        $ 1403 "Direction: Base Z+"
        global move_thread_flag_1403=0
        thread move_thread_1403():
          enter_critical
          move_thread_flag_1403 = 1
          local towardsPos=calculate_point_to_move_towards(p[0.0,0.0,0.0,0.0,0.0,0.0], [0.0,0.0,1.0], 0.05)
          movel(towardsPos, a=0.04, v=0.03)
          move_thread_flag_1403 = 2
          exit_critical
        end
        move_thread_flag_1403 = 0
        move_thread_han_1403 = run move_thread_1403()
        while (True):
          sleep(1.0E-10)
          if (move_thread_flag_1403 > 1):
            join move_thread_han_1403
            $ 1404 "Until (distance)"
            break
          end
          sync()
        end
        $ 1405 "MoveJ"
        $ 1406 "internos" "breakAfter"
        movej(internos, a=1.3962634015954636, v=1.0471975511965976)
        $ 1407 "Wait: 0.3"
        sleep(0.3)
        $ 1408 "Set CO[1]=Apagar"
        set_configurable_digital_out(1, False)
        $ 1409 "Wait: 0.3"
        sleep(0.3)
        $ 1410 "If barrenoActual≟13"
        if (barrenoActual == 13):
          $ 1411 "Direction: Base Z+"
          global move_thread_flag_1411=0
          thread move_thread_1411():
            enter_critical
            move_thread_flag_1411 = 1
            local towardsPos=calculate_point_to_move_towards(p[0.0,0.0,0.0,0.0,0.0,0.0], [0.0,0.0,1.0], 0.03)
            movel(towardsPos, a=1.2, v=0.25)
            move_thread_flag_1411 = 2
            exit_critical
          end
          move_thread_flag_1411 = 0
          move_thread_han_1411 = run move_thread_1411()
          while (True):
            sleep(1.0E-10)
            if (move_thread_flag_1411 > 1):
              join move_thread_han_1411
              $ 1412 "Until (distance)"
              break
            end
            sync()
          end
          $ 1413 "MoveJ"
          $ 1414 "Zona_izq1" "breakAfter"
          movej(get_inverse_kin(Zona_izq1_p, qnear=Zona_izq1_q), a=1.3962634015954636, v=1.0471975511965976)
          $ 1415 "Posicion_Cero" "breakAfter"
          movej(get_inverse_kin(Posicion_Cero_p, qnear=Posicion_Cero_q), a=1.3962634015954636, v=1.0471975511965976)
          $ 1416 "Call Quitar_Broca_Chida"
          Quitar_Broca_Chida()
          $ 1417 "Call Poner_Broca"
          Poner_Broca()
          $ 1418 "MoveJ"
          $ 1419 "Posicion_Cero" "breakAfter"
          movej(get_inverse_kin(Posicion_Cero_p, qnear=Posicion_Cero_q), a=1.3962634015954636, v=1.0471975511965976)
          $ 1420 "Zona_izq1" "breakAfter"
          movej(get_inverse_kin(Zona_izq1_p, qnear=Zona_izq1_q), a=1.3962634015954636, v=1.0471975511965976)
        else:
          $ 1421 "ElseIf barrenoActual≟27"
          if (barrenoActual == 27):
            $ 1422 "Direction: Base Z+"
            global move_thread_flag_1422=0
            thread move_thread_1422():
              enter_critical
              move_thread_flag_1422 = 1
              local towardsPos=calculate_point_to_move_towards(p[0.0,0.0,0.0,0.0,0.0,0.0], [0.0,0.0,1.0], 0.03)
              movel(towardsPos, a=1.2, v=0.25)
              move_thread_flag_1422 = 2
              exit_critical
            end
            move_thread_flag_1422 = 0
            move_thread_han_1422 = run move_thread_1422()
            while (True):
              sleep(1.0E-10)
              if (move_thread_flag_1422 > 1):
                join move_thread_han_1422
                $ 1423 "Until (distance)"
                break
              end
              sync()
            end
            $ 1424 "MoveJ"
            $ 1425 "Zona_izq1" "breakAfter"
            movej(get_inverse_kin(Zona_izq1_p, qnear=Zona_izq1_q), a=1.3962634015954636, v=1.0471975511965976)
            $ 1426 "Posicion_Cero" "breakAfter"
            movej(get_inverse_kin(Posicion_Cero_p, qnear=Posicion_Cero_q), a=1.3962634015954636, v=1.0471975511965976)
            $ 1427 "Call Quitar_Broca_Chida"
            Quitar_Broca_Chida()
            $ 1428 "Set carrusel_home=Encender"
            modbus_set_output_signal("carrusel_home", True)
            $ 1429 "Wait: 1.0"
            sleep(1.0)
            $ 1430 "Set carrusel_home=Apagar"
            modbus_set_output_signal("carrusel_home", False)
            $ 1431 "Set mensaje_mw10=85"
            modbus_set_output_register("mensaje_mw10", 85)
            $ 1432 "Wait Continuar_M30=HI"
            while (modbus_get_signal_status("Continuar_M30") == False):
              sync()
            end
            $ 1433 "Wait: 1.0"
            sleep(1.0)
            $ 1434 "Set mensaje_mw10=120"
            modbus_set_output_register("mensaje_mw10", 120)
            $ 1435 "Wait Continuar_M30=HI"
            while (modbus_get_signal_status("Continuar_M30") == False):
              sync()
            end
            $ 1436 "Wait: 1.0"
            sleep(1.0)
            $ 1437 "Set carrusel_home=Encender"
            modbus_set_output_signal("carrusel_home", True)
            $ 1438 "Wait: 1.0"
            sleep(1.0)
            $ 1439 "Set carrusel_home=Apagar"
            modbus_set_output_signal("carrusel_home", False)
            $ 1440 "Set mensaje_mw10=90"
            modbus_set_output_register("mensaje_mw10", 90)
            $ 1441 "Wait Continuar_M30=HI"
            while (modbus_get_signal_status("Continuar_M30") == False):
              sync()
            end
            $ 1442 "Wait: 1.0"
            sleep(1.0)
            $ 1443 "Call Poner_Broca"
            Poner_Broca()
            $ 1444 "broca≔217"
            global broca=217
            $ 1445 "MoveJ"
            $ 1446 "Posicion_Cero" "breakAfter"
            movej(get_inverse_kin(Posicion_Cero_p, qnear=Posicion_Cero_q), a=1.3962634015954636, v=1.0471975511965976)
            $ 1447 "Zona_izq1" "breakAfter"
            movej(get_inverse_kin(Zona_izq1_p, qnear=Zona_izq1_q), a=1.3962634015954636, v=1.0471975511965976)
            $ 1448 "Set mensaje_mw10=95"
            modbus_set_output_register("mensaje_mw10", 95)
            $ 1449 "Wait Continuar_M30=HI"
            while (modbus_get_signal_status("Continuar_M30") == False):
              sync()
            end
            $ 1450 "Wait: 1.0"
            sleep(1.0)
            $ 1451 "Set mensaje_mw10=150"
            modbus_set_output_register("mensaje_mw10", 150)
            $ 1452 "Wait Continuar_M30=HI"
            while (modbus_get_signal_status("Continuar_M30") == False):
              sync()
            end
            $ 1453 "Wait: 1.0"
            sleep(1.0)
          end
        end
        $ 1454 "barrenoActual≔barrenoActual+1"
        global barrenoActual=barrenoActual+1
      end
      $ 1455 "Linea 1 a 217"
      $ 1456 "broca≔217"
      global broca=217
      $ 1457 "Buje_inicial"
      $ 1458 "Buje_Inicial≔L1B2"
      global Buje_Inicial=L1B2
      $ 1459 "Buje_final"
      $ 1460 "Buje_Final≔L1B1"
      global Buje_Final=L1B1
      $ 1461 "barrenosTotales≔27"
      global barrenosTotales=27
      $ 1462 "barrenoActual≔1"
      global barrenoActual=1
      $ 1463 "Loop barrenoActual≤barrenosTotales"
      while (barrenoActual <= barrenosTotales):
        $ 1464 "MoveL"
        $ 1465 "bajada_broca≔p[0,0,0.018,0,0,0]"
        global bajada_broca=p[0,0,0.018,0,0,0]
        $ 1466 "internos≔interpolate_pose(Buje_Inicial, Buje_Final, ((barrenoActual)-1)/((barrenosTotales)-1))"
        global internos= interpolate_pose (Buje_Inicial, Buje_Final, ((barrenoActual)-1)/((barrenosTotales)-1))
        $ 1467 "Alturas"
        $ 1468 "If barrenoActual≟3 or barrenoActual≟5 or barrenoActual≟7 or barrenoActual≟9 or barrenoActual≟11 or barrenoActual≟13 or barrenoActual≟15 or barrenoActual≟17 or barrenoActual≟19 or barrenoActual≟21 or barrenoActual≟23 or barrenoActual≟25 or barrenoActual≟27 or barrenoActual≟1"
        if (barrenoActual == 3  or  barrenoActual == 5  or  barrenoActual == 7  or  barrenoActual == 9  or  barrenoActual == 11  or  barrenoActual == 13  or  barrenoActual == 15  or  barrenoActual == 17  or  barrenoActual == 19  or  barrenoActual == 21  or  barrenoActual == 23  or  barrenoActual == 25  or  barrenoActual == 27  or  barrenoActual == 1):
          $ 1469 "Set mensaje_mw10=200"
          modbus_set_output_register("mensaje_mw10", 200)
          $ 1470 "Wait Continuar_M30=HI"
          while (modbus_get_signal_status("Continuar_M30") == False):
            sync()
          end
          $ 1471 "Wait: 1.0"
          sleep(1.0)
          $ 1472 "Set mensaje_mw10=150"
          modbus_set_output_register("mensaje_mw10", 150)
          $ 1473 "Wait: 1.0"
          sleep(1.0)
        end
        $ 1474 "MoveJ"
        $ 1475 "internos" "breakAfter"
        movej(internos, a=1.3962634015954636, v=1.0471975511965976)
        $ 1476 "Wait: 2.0"
        sleep(2.0)
        $ 1477 "If P1h[2]<P2h[2]"
        if (P1h[2]<P2h[2]):
          $ 1478 "acomodin≔(altura/(barrenosTotales-1))*(barrenoActual-1)"
          global acomodin=(altura/(barrenosTotales-1))*(barrenoActual-1)
          $ 1479 "tcp_chido≔get_actual_tcp_pose()"
          global tcp_chido= get_actual_tcp_pose ()
          $ 1480 "offset_bajada≔p[tcp_chido[0],tcp_chido[1],((alta-0.0095)-(acomodin/1000)),tcp_chido[3],tcp_chido[4],tcp_chido[5]]"
          global offset_bajada=p[tcp_chido[0],tcp_chido[1],((alta-0.0095)-(acomodin/1000)),tcp_chido[3],tcp_chido[4],tcp_chido[5]]
          $ 1481 "MoveL"
          $ 1482 "offset_bajada" "breakAfter"
          movel(offset_bajada, a=0.03, v=0.015)
        else:
          $ 1483 "Else" "noBreak"
          $ 1484 "acomodin≔(altura/(barrenosTotales-1))*(26-(barrenoActual-1))"
          global acomodin=(altura/(barrenosTotales-1))*(26-(barrenoActual-1))
          $ 1485 "tcp_chido≔get_actual_tcp_pose()"
          global tcp_chido= get_actual_tcp_pose ()
          $ 1486 "offset_bajada≔p[tcp_chido[0],tcp_chido[1],((alta-0.0095)-(acomodin/1000)),tcp_chido[3],tcp_chido[4],tcp_chido[5]]"
          global offset_bajada=p[tcp_chido[0],tcp_chido[1],((alta-0.0095)-(acomodin/1000)),tcp_chido[3],tcp_chido[4],tcp_chido[5]]
          $ 1487 "MoveL"
          $ 1488 "offset_bajada" "breakAfter"
          movel(offset_bajada, a=0.03, v=0.015)
        end
        $ 1489 "Freemove"
        $ 1490 "Wait: 2.0"
        sleep(2.0)
        $ 1491 "freedrive_mode()"
        freedrive_mode()
        $ 1492 "Wait: 2.5"
        sleep(2.5)
        $ 1493 "end_freedrive_mode()"
        end_freedrive_mode()
        $ 1494 "Wait: 0.3"
        sleep(0.3)
        $ 1495 "Set CO[1]=Encender"
        set_configurable_digital_out(1, True)
        $ 1496 "Wait: 1.0"
        sleep(1.0)
        $ 1497 "Wait: 0.3"
        sleep(0.3)
        $ 1498 "Wait: 0.3"
        sleep(0.3)
        $ 1499 "Wait: 0.3"
        sleep(0.3)
        $ 1500 "Loop 1 times"
        Loop_76 = 0
        while (Loop_76 < 1):
          $ 1501 "Poses_taladrado≔pose_sub(get_actual_tcp_pose(), bajada_broca)"
          global Poses_taladrado= pose_sub ( get_actual_tcp_pose (), bajada_broca)
          $ 1502 "Poses_taladrado" "breakAfter"
          movel(Poses_taladrado, a=0.005, v=0.001)
          $ 1503 "If bajada_broca≟p[0,0,0.018,0,0,0]"
          if (bajada_broca == p[0,0,0.018,0,0,0]):
            $ 1504 "num_barreno≔str_cat('Barreno: ',barrenoActual)"
            global num_barreno=str_cat("Barreno: ",barrenoActual)
            $ 1505 "tcp_actual≔get_actual_tcp_pose()"
            global tcp_actual= get_actual_tcp_pose ()
            $ 1506 "X_actual≔str_cat('     X: ',tcp_actual[0])"
            global X_actual=str_cat("     X: ",tcp_actual[0])
            $ 1507 "Y_actual≔str_cat('     Y: ',tcp_actual[1])"
            global Y_actual=str_cat("     Y: ",tcp_actual[1])
            $ 1508 "pos_barreno≔str_cat(X_actual,Y_actual)"
            global pos_barreno=str_cat(X_actual,Y_actual)
            $ 1509 "textmsg(num_barreno,pos_barreno)"
            textmsg(num_barreno,pos_barreno)
          end
          $ 1510 "Poses_taladrado≔pose_add(get_actual_tcp_pose(), bajada_broca)"
          global Poses_taladrado= pose_add ( get_actual_tcp_pose (), bajada_broca)
          $ 1511 "Poses_taladrado" "breakAfter"
          movel(Poses_taladrado, a=0.01, v=0.01)
          $ 1512 "bajada_broca≔pose_add(bajada_broca, p[0,0,0.018,0,0,0])"
          global bajada_broca= pose_add (bajada_broca, p[0,0,0.018,0,0,0])
          Loop_76 = Loop_76 + 1
        end
        $ 1513 "Direction: Base Z+"
        global move_thread_flag_1513=0
        thread move_thread_1513():
          enter_critical
          move_thread_flag_1513 = 1
          local towardsPos=calculate_point_to_move_towards(p[0.0,0.0,0.0,0.0,0.0,0.0], [0.0,0.0,1.0], 0.05)
          movel(towardsPos, a=0.04, v=0.03)
          move_thread_flag_1513 = 2
          exit_critical
        end
        move_thread_flag_1513 = 0
        move_thread_han_1513 = run move_thread_1513()
        while (True):
          sleep(1.0E-10)
          if (move_thread_flag_1513 > 1):
            join move_thread_han_1513
            $ 1514 "Until (distance)"
            break
          end
          sync()
        end
        $ 1515 "MoveJ"
        $ 1516 "internos" "breakAfter"
        movej(internos, a=1.3962634015954636, v=1.0471975511965976)
        $ 1517 "Wait: 0.3"
        sleep(0.3)
        $ 1518 "Set CO[1]=Apagar"
        set_configurable_digital_out(1, False)
        $ 1519 "Wait: 0.3"
        sleep(0.3)
        $ 1520 "If barrenoActual≟13 or barrenoActual≟27"
        if (barrenoActual == 13  or  barrenoActual == 27):
          $ 1521 "Direction: Base Z+"
          global move_thread_flag_1521=0
          thread move_thread_1521():
            enter_critical
            move_thread_flag_1521 = 1
            local towardsPos=calculate_point_to_move_towards(p[0.0,0.0,0.0,0.0,0.0,0.0], [0.0,0.0,1.0], 0.03)
            movel(towardsPos, a=1.2, v=0.25)
            move_thread_flag_1521 = 2
            exit_critical
          end
          move_thread_flag_1521 = 0
          move_thread_han_1521 = run move_thread_1521()
          while (True):
            sleep(1.0E-10)
            if (move_thread_flag_1521 > 1):
              join move_thread_han_1521
              $ 1522 "Until (distance)"
              break
            end
            sync()
          end
          $ 1523 "MoveJ"
          $ 1524 "Zona_izq1" "breakAfter"
          movej(get_inverse_kin(Zona_izq1_p, qnear=Zona_izq1_q), a=1.3962634015954636, v=1.0471975511965976)
          $ 1525 "Posicion_Cero" "breakAfter"
          movej(get_inverse_kin(Posicion_Cero_p, qnear=Posicion_Cero_q), a=1.3962634015954636, v=1.0471975511965976)
          $ 1526 "Call Quitar_Broca_Chida"
          Quitar_Broca_Chida()
          $ 1527 "Call Poner_Broca"
          Poner_Broca()
          $ 1528 "MoveJ"
          $ 1529 "Posicion_Cero" "breakAfter"
          movej(get_inverse_kin(Posicion_Cero_p, qnear=Posicion_Cero_q), a=1.3962634015954636, v=1.0471975511965976)
          $ 1530 "Zona_izq1" "breakAfter"
          movej(get_inverse_kin(Zona_izq1_p, qnear=Zona_izq1_q), a=1.3962634015954636, v=1.0471975511965976)
        end
        $ 1531 "barrenoActual≔barrenoActual+1"
        global barrenoActual=barrenoActual+1
      end
      $ 1532 "Linea 2 a 217"
      $ 1533 "broca≔217"
      global broca=217
      $ 1534 "Buje_inicial"
      $ 1535 "Buje_Inicial≔L2B2"
      global Buje_Inicial=L2B2
      $ 1536 "Buje_final"
      $ 1537 "Buje_Final≔L2B1"
      global Buje_Final=L2B1
      $ 1538 "barrenosTotales≔27"
      global barrenosTotales=27
      $ 1539 "barrenoActual≔1"
      global barrenoActual=1
      $ 1540 "Loop barrenoActual≤barrenosTotales"
      while (barrenoActual <= barrenosTotales):
        $ 1541 "MoveL"
        $ 1542 "bajada_broca≔p[0,0,0.018,0,0,0]"
        global bajada_broca=p[0,0,0.018,0,0,0]
        $ 1543 "internos≔interpolate_pose(Buje_Inicial, Buje_Final, ((barrenoActual)-1)/((barrenosTotales)-1))"
        global internos= interpolate_pose (Buje_Inicial, Buje_Final, ((barrenoActual)-1)/((barrenosTotales)-1))
        $ 1544 "Alturas"
        $ 1545 "If barrenoActual≟3 or barrenoActual≟5 or barrenoActual≟7 or barrenoActual≟9 or barrenoActual≟11 or barrenoActual≟13 or barrenoActual≟15 or barrenoActual≟17 or barrenoActual≟19 or barrenoActual≟21 or barrenoActual≟23 or barrenoActual≟25 or barrenoActual≟27 or barrenoActual≟1"
        if (barrenoActual == 3  or  barrenoActual == 5  or  barrenoActual == 7  or  barrenoActual == 9  or  barrenoActual == 11  or  barrenoActual == 13  or  barrenoActual == 15  or  barrenoActual == 17  or  barrenoActual == 19  or  barrenoActual == 21  or  barrenoActual == 23  or  barrenoActual == 25  or  barrenoActual == 27  or  barrenoActual == 1):
          $ 1546 "Set mensaje_mw10=200"
          modbus_set_output_register("mensaje_mw10", 200)
          $ 1547 "Wait Continuar_M30=HI"
          while (modbus_get_signal_status("Continuar_M30") == False):
            sync()
          end
          $ 1548 "Wait: 1.0"
          sleep(1.0)
          $ 1549 "Set mensaje_mw10=150"
          modbus_set_output_register("mensaje_mw10", 150)
          $ 1550 "Wait: 1.0"
          sleep(1.0)
        end
        $ 1551 "MoveJ"
        $ 1552 "internos" "breakAfter"
        movej(internos, a=1.3962634015954636, v=1.0471975511965976)
        $ 1553 "Wait: 2.0"
        sleep(2.0)
        $ 1554 "If P1h[2]<P2h[2]"
        if (P1h[2]<P2h[2]):
          $ 1555 "acomodin≔(altura/(barrenosTotales-1))*(barrenoActual-1)"
          global acomodin=(altura/(barrenosTotales-1))*(barrenoActual-1)
          $ 1556 "tcp_chido≔get_actual_tcp_pose()"
          global tcp_chido= get_actual_tcp_pose ()
          $ 1557 "offset_bajada≔p[tcp_chido[0],tcp_chido[1],((alta-0.0095)-(acomodin/1000)),tcp_chido[3],tcp_chido[4],tcp_chido[5]]"
          global offset_bajada=p[tcp_chido[0],tcp_chido[1],((alta-0.0095)-(acomodin/1000)),tcp_chido[3],tcp_chido[4],tcp_chido[5]]
          $ 1558 "MoveL"
          $ 1559 "offset_bajada" "breakAfter"
          movel(offset_bajada, a=0.03, v=0.015)
        else:
          $ 1560 "Else" "noBreak"
          $ 1561 "acomodin≔(altura/(barrenosTotales-1))*(26-(barrenoActual-1))"
          global acomodin=(altura/(barrenosTotales-1))*(26-(barrenoActual-1))
          $ 1562 "tcp_chido≔get_actual_tcp_pose()"
          global tcp_chido= get_actual_tcp_pose ()
          $ 1563 "offset_bajada≔p[tcp_chido[0],tcp_chido[1],((alta-0.0095)-(acomodin/1000)),tcp_chido[3],tcp_chido[4],tcp_chido[5]]"
          global offset_bajada=p[tcp_chido[0],tcp_chido[1],((alta-0.0095)-(acomodin/1000)),tcp_chido[3],tcp_chido[4],tcp_chido[5]]
          $ 1564 "MoveL"
          $ 1565 "offset_bajada" "breakAfter"
          movel(offset_bajada, a=0.03, v=0.015)
        end
        $ 1566 "Freemove"
        $ 1567 "Wait: 2.0"
        sleep(2.0)
        $ 1568 "freedrive_mode()"
        freedrive_mode()
        $ 1569 "Wait: 2.5"
        sleep(2.5)
        $ 1570 "end_freedrive_mode()"
        end_freedrive_mode()
        $ 1571 "Wait: 0.3"
        sleep(0.3)
        $ 1572 "Set CO[1]=Encender"
        set_configurable_digital_out(1, True)
        $ 1573 "Wait: 1.0"
        sleep(1.0)
        $ 1574 "Wait: 0.3"
        sleep(0.3)
        $ 1575 "Wait: 0.3"
        sleep(0.3)
        $ 1576 "Wait: 0.3"
        sleep(0.3)
        $ 1577 "Loop 1 times"
        Loop_78 = 0
        while (Loop_78 < 1):
          $ 1578 "Poses_taladrado≔pose_sub(get_actual_tcp_pose(), bajada_broca)"
          global Poses_taladrado= pose_sub ( get_actual_tcp_pose (), bajada_broca)
          $ 1579 "Poses_taladrado" "breakAfter"
          movel(Poses_taladrado, a=0.005, v=0.001)
          $ 1580 "If bajada_broca≟p[0,0,0.018,0,0,0]"
          if (bajada_broca == p[0,0,0.018,0,0,0]):
            $ 1581 "num_barreno≔str_cat('Barreno: ',barrenoActual)"
            global num_barreno=str_cat("Barreno: ",barrenoActual)
            $ 1582 "tcp_actual≔get_actual_tcp_pose()"
            global tcp_actual= get_actual_tcp_pose ()
            $ 1583 "X_actual≔str_cat('     X: ',tcp_actual[0])"
            global X_actual=str_cat("     X: ",tcp_actual[0])
            $ 1584 "Y_actual≔str_cat('     Y: ',tcp_actual[1])"
            global Y_actual=str_cat("     Y: ",tcp_actual[1])
            $ 1585 "pos_barreno≔str_cat(X_actual,Y_actual)"
            global pos_barreno=str_cat(X_actual,Y_actual)
            $ 1586 "textmsg(num_barreno,pos_barreno)"
            textmsg(num_barreno,pos_barreno)
          end
          $ 1587 "Poses_taladrado≔pose_add(get_actual_tcp_pose(), bajada_broca)"
          global Poses_taladrado= pose_add ( get_actual_tcp_pose (), bajada_broca)
          $ 1588 "Poses_taladrado" "breakAfter"
          movel(Poses_taladrado, a=0.01, v=0.01)
          $ 1589 "bajada_broca≔pose_add(bajada_broca, p[0,0,0.018,0,0,0])"
          global bajada_broca= pose_add (bajada_broca, p[0,0,0.018,0,0,0])
          Loop_78 = Loop_78 + 1
        end
        $ 1590 "Direction: Base Z+"
        global move_thread_flag_1590=0
        thread move_thread_1590():
          enter_critical
          move_thread_flag_1590 = 1
          local towardsPos=calculate_point_to_move_towards(p[0.0,0.0,0.0,0.0,0.0,0.0], [0.0,0.0,1.0], 0.05)
          movel(towardsPos, a=0.04, v=0.03)
          move_thread_flag_1590 = 2
          exit_critical
        end
        move_thread_flag_1590 = 0
        move_thread_han_1590 = run move_thread_1590()
        while (True):
          sleep(1.0E-10)
          if (move_thread_flag_1590 > 1):
            join move_thread_han_1590
            $ 1591 "Until (distance)"
            break
          end
          sync()
        end
        $ 1592 "MoveJ"
        $ 1593 "internos" "breakAfter"
        movej(internos, a=1.3962634015954636, v=1.0471975511965976)
        $ 1594 "Wait: 0.3"
        sleep(0.3)
        $ 1595 "Set CO[1]=Apagar"
        set_configurable_digital_out(1, False)
        $ 1596 "Wait: 0.3"
        sleep(0.3)
        $ 1597 "If barrenoActual≟13"
        if (barrenoActual == 13):
          $ 1598 "Direction: Base Z+"
          global move_thread_flag_1598=0
          thread move_thread_1598():
            enter_critical
            move_thread_flag_1598 = 1
            local towardsPos=calculate_point_to_move_towards(p[0.0,0.0,0.0,0.0,0.0,0.0], [0.0,0.0,1.0], 0.03)
            movel(towardsPos, a=1.2, v=0.25)
            move_thread_flag_1598 = 2
            exit_critical
          end
          move_thread_flag_1598 = 0
          move_thread_han_1598 = run move_thread_1598()
          while (True):
            sleep(1.0E-10)
            if (move_thread_flag_1598 > 1):
              join move_thread_han_1598
              $ 1599 "Until (distance)"
              break
            end
            sync()
          end
          $ 1600 "MoveJ"
          $ 1601 "Zona_izq1" "breakAfter"
          movej(get_inverse_kin(Zona_izq1_p, qnear=Zona_izq1_q), a=1.3962634015954636, v=1.0471975511965976)
          $ 1602 "Posicion_Cero" "breakAfter"
          movej(get_inverse_kin(Posicion_Cero_p, qnear=Posicion_Cero_q), a=1.3962634015954636, v=1.0471975511965976)
          $ 1603 "Call Quitar_Broca_Chida"
          Quitar_Broca_Chida()
          $ 1604 "Call Poner_Broca"
          Poner_Broca()
          $ 1605 "MoveJ"
          $ 1606 "Posicion_Cero" "breakAfter"
          movej(get_inverse_kin(Posicion_Cero_p, qnear=Posicion_Cero_q), a=1.3962634015954636, v=1.0471975511965976)
          $ 1607 "Zona_izq1" "breakAfter"
          movej(get_inverse_kin(Zona_izq1_p, qnear=Zona_izq1_q), a=1.3962634015954636, v=1.0471975511965976)
        else:
          $ 1608 "ElseIf barrenoActual≟27"
          if (barrenoActual == 27):
            $ 1609 "Direction: Base Z+"
            global move_thread_flag_1609=0
            thread move_thread_1609():
              enter_critical
              move_thread_flag_1609 = 1
              local towardsPos=calculate_point_to_move_towards(p[0.0,0.0,0.0,0.0,0.0,0.0], [0.0,0.0,1.0], 0.03)
              movel(towardsPos, a=1.2, v=0.25)
              move_thread_flag_1609 = 2
              exit_critical
            end
            move_thread_flag_1609 = 0
            move_thread_han_1609 = run move_thread_1609()
            while (True):
              sleep(1.0E-10)
              if (move_thread_flag_1609 > 1):
                join move_thread_han_1609
                $ 1610 "Until (distance)"
                break
              end
              sync()
            end
            $ 1611 "MoveJ"
            $ 1612 "Zona_izq1" "breakAfter"
            movej(get_inverse_kin(Zona_izq1_p, qnear=Zona_izq1_q), a=1.3962634015954636, v=1.0471975511965976)
            $ 1613 "Posicion_Cero" "breakAfter"
            movej(get_inverse_kin(Posicion_Cero_p, qnear=Posicion_Cero_q), a=1.3962634015954636, v=1.0471975511965976)
            $ 1614 "Call Quitar_Broca_Chida"
            Quitar_Broca_Chida()
            $ 1615 "Set carrusel_home=Encender"
            modbus_set_output_signal("carrusel_home", True)
            $ 1616 "Wait: 1.0"
            sleep(1.0)
            $ 1617 "Set carrusel_home=Apagar"
            modbus_set_output_signal("carrusel_home", False)
            $ 1618 "Set mensaje_mw10=120"
            modbus_set_output_register("mensaje_mw10", 120)
            $ 1619 "Wait Continuar_M30=HI"
            while (modbus_get_signal_status("Continuar_M30") == False):
              sync()
            end
            $ 1620 "Wait: 1.0"
            sleep(1.0)
            $ 1621 "Set mensaje_mw10=100"
            modbus_set_output_register("mensaje_mw10", 100)
            $ 1622 "Wait Continuar_M30=HI"
            while (modbus_get_signal_status("Continuar_M30") == False):
              sync()
            end
            $ 1623 "Wait: 1.0"
            sleep(1.0)
            $ 1624 "MoveJ"
            $ 1625 "Traslacion_izq" "breakAfter"
            movej(get_inverse_kin(Traslacion_izq_p, qnear=Traslacion_izq_q), a=1.3962634015954636, v=1.0471975511965976)
          end
        end
        $ 1626 "barrenoActual≔barrenoActual+1"
        global barrenoActual=barrenoActual+1
      end
      $ 1628 "Traslacion"
      $ 1629 "MoveJ"
      $ 1630 "Traslacion_izq" "breakAfter"
      movej(get_inverse_kin(Traslacion_izq_p, qnear=Traslacion_izq_q), a=1.3962634015954636, v=1.0471975511965976)
      $ 1631 "Set mensaje_mw10=105"
      modbus_set_output_register("mensaje_mw10", 105)
      $ 1632 "Wait Continuar_M30=HI"
      while (modbus_get_signal_status("Continuar_M30") == False):
        sync()
      end
      $ 1633 "Wait: 1.0"
      sleep(1.0)
      $ 1634 "Set mensaje_mw10=110"
      modbus_set_output_register("mensaje_mw10", 110)
      $ 1635 "Wait Continuar_M30=HI"
      while (modbus_get_signal_status("Continuar_M30") == False):
        sync()
      end
      $ 1636 "Wait: 1.0"
      sleep(1.0)
      $ 1637 "Set postrnas_m187=Encender"
      modbus_set_output_signal("postrnas_m187", True)
      $ 1638 "Wait: 1.0"
      sleep(1.0)
      $ 1639 "Set Home_M20=Encender"
      modbus_set_output_signal("Home_M20", True)
      $ 1640 "Wait: 1.0"
      sleep(1.0)
      $ 1641 "Set Home_M20=Apagar"
      modbus_set_output_signal("Home_M20", False)
      $ 1642 "Set postrnas_m187=Apagar"
      modbus_set_output_signal("postrnas_m187", False)
      $ 1643 "Wait: 5.0"
      sleep(5.0)
      $ 1644 "Apagar"
      $ 1645 "Set mensaje_mw10=115"
      modbus_set_output_register("mensaje_mw10", 115)
      $ 1646 "Wait Continuar_M30=HI"
      while (modbus_get_signal_status("Continuar_M30") == False):
        sync()
      end
      $ 1647 "Wait: 1.0"
      sleep(1.0)
      $ 1648 "MoveJ"
      $ 1649 "Waypoint_9" "breakAfter"
      movej(get_inverse_kin(Waypoint_9_p, qnear=Waypoint_9_q), a=1.3962634015954636, v=1.0471975511965976)
      $ 1650 "Waypoint_8" "breakAfter"
      movej(get_inverse_kin(Waypoint_8_p, qnear=Waypoint_8_q), a=1.3962634015954636, v=1.0471975511965976)
      $ 1651 "Off_izquierda" "breakAfter"
      movej(get_inverse_kin(Off_izquierda_p, qnear=Off_izquierda_q), a=1.3962634015954636, v=1.0471975511965976)
      $ 1652 "Set mensaje_mw10=0"
      modbus_set_output_register("mensaje_mw10", 0)
      $ 1653 "Wait: 1.0"
      sleep(1.0)
      $ 1654 "Wait Continuar_M30=HI"
      while (modbus_get_signal_status("Continuar_M30") == False):
        sync()
      end
      $ 1655 "Wait: 1.0"
      sleep(1.0)
      $ 1656 "Popup: DAS apagado"
      popup("DAS apagado", "Advertencia", True, False, blocking=False)
      halt
    else:
      $ 1657 "ElseIf Lado_Correr≟2"
      if (modbus_get_signal_status("Lado_Correr") == 2):
        $ 1658 "Popup: Apagar DAS"
        popup("Apagar DAS", "Advertencia", True, False, blocking=False)
        halt
      else:
        $ 1659 "ElseIf Lado_Correr≟3"
        if (modbus_get_signal_status("Lado_Correr") == 3):
          $ 1660 "Popup: Apagar DAS"
          popup("Apagar DAS", "Advertencia", True, False, blocking=False)
          halt
        else:
          $ 1661 "Else" "noBreak"
          $ 1662 "Lado≔ False "
          global Lado=  False
          $ 1663 "Popup: DAS no anclado"
          popup("DAS no anclado", "Advertencia", True, False, blocking=False)
          halt
        end
      end
    end
  end
end
